// TIA Portal V18 export
VAR_GLOBAL   // PLC tag table "19_AE1-SA3"
   "iAE1-SA3p" AT %I12.0 : Bool;   // 5
   "iAE1-SA3" AT %I12.1 : Bool;   // 5
   "iAE1-SA3a" AT %I17.6 : Bool;
   "oAE1-SA3p" AT %Q9.3 : Bool;
   "oAE1-SA3" AT %Q9.4 : Bool;
END_VAR
